{attribute 'GeneratedUsingTerminal: EL2502-0000-0016'}
{attribute addProperty BoxType "EL2502-0000-0016"}
{attribute addProperty Id "PWM_outputAT %Q*UINT2"}
{attribute addProperty CRC "1281526221"}
{attribute addProperty Size "2"}
TYPE PWM_Outputs_Channel_4C6289CD :
STRUCT
	{attribute addProperty Name "PWM_output"}
	PWM_output AT %Q* : UINT;
END_STRUCT
END_TYPE

(* stored: Version 1.2.0.0, ProductVersion 3.1.4024.9
   DUT PWM_Outputs_Channel_4C6289CD: Id {cb0227bc-2f05-4765-972f-9e3025e41385} *)
